{attribute 'no_explicit_call' := 'do not call this function block directly'} 
FUNCTION_BLOCK RenameFile EXTENDS ToolkitObject IMPLEMENTS IAction
VAR
	{attribute 'OPC.UA.DA' := '0'}
	_ClassName : STRING := __POUNAME();

	{attribute 'OPC.UA.DA' := '0'}
    _Rename : Tc2_System.FB_FileRename;
	
	{attribute 'OPC.UA.DA' := '0'}
	_NeedStart : BOOL;
	{attribute 'OPC.UA.DA' := '0'}
	_Done : BOOL;
END_VAR

{attribute 'monitoring' := 'call'}
{attribute 'OPC.UA.DA.Property' := '1'}
{attribute 'OPC.UA.DA' := '1'}
PROPERTY AmsNetId : Tc2_System.T_AmsNetID
GET
AmsNetId := _Rename.sNetId;
END_GET
SET
_Rename.sNetId := AmsNetId;
END_SET
END_PROPERTY

{attribute 'monitoring' := 'call'}
{attribute 'OPC.UA.DA.Property' := '1'}
{attribute 'OPC.UA.DA.Access' := '1'}
PROPERTY Busy : BOOL
GET
Busy := _NeedStart OR_ELSE _Rename.bBusy;
END_GET
END_PROPERTY

{attribute 'monitoring' := 'call'}
PROPERTY ClassName : STRING
GET
ClassName := _ClassName;
END_GET
END_PROPERTY

{attribute 'monitoring' := 'call'}
{attribute 'OPC.UA.DA.Property' := '1'}
{attribute 'OPC.UA.DA.Access' := '1'}
PROPERTY Done : BOOL
GET
Done := _Done;
END_GET
END_PROPERTY

{attribute 'monitoring' := 'call'}
{attribute 'OPC.UA.DA.Property' := '1'}
{attribute 'OPC.UA.DA.Access' := '1'}
PROPERTY Error : BOOL
GET
Error := _Rename.bError;
END_GET
END_PROPERTY

METHOD Execute
VAR
	message : ERROR_MESSAGE;
END_VAR
IF _NeedStart OR_ELSE _Rename.bBusy THEN
	_Rename(bExecute := TRUE);
	_NeedStart := FALSE;
	
	IF _Rename.bError THEN
		message := "An error occurred while renaming the file '";
		WStringHelper.Append6(message, TO_WSTRING(_Rename.sOldName), "' to '", TO_WSTRING(_Rename.sNewName), " in directory '", TO_WSTRING(_Rename.ePath), "'");	
		_LastException.Configure(message, __POUNAME(), ClassName, CurrentNamespace.Name, __POSITION(), _Rename.nErrId);
	ELSIF NOT _Rename.bBusy THEN
		_Done := TRUE;
	END_IF
END_IF
END_METHOD

{attribute 'monitoring' := 'call'}
{attribute 'OPC.UA.DA.Property' := '1'}
{attribute 'OPC.UA.DA.Access' := '1'}
PROPERTY LastException : REFERENCE TO Exception
GET
LastException REF= _LastException;
END_GET
END_PROPERTY

{attribute 'monitoring' := 'call'}
{attribute 'OPC.UA.DA.Property' := '1'}
{attribute 'OPC.UA.DA' := '1'}
PROPERTY PathType : Tc2_System.E_OpenPath
GET
PathType := _Rename.ePath;
END_GET
SET
_Rename.ePath := PathType;
END_SET
END_PROPERTY

METHOD Start
VAR_INPUT
	oldFilePath : Tc2_System.T_MaxString;
	newFilePath : Tc2_System.T_MaxString;
END_VAR
_NeedStart := TRUE;
_Done := FALSE;
_Rename.sOldName := oldFilePath;
_Rename.sNewName := newFilePath;

_LastException.Clear();
END_METHOD

{attribute 'monitoring' := 'call'}
{attribute 'OPC.UA.DA.Property' := '1'}
{attribute 'OPC.UA.DA' := '1'}
PROPERTY Timeout : TIME
GET
Timeout := _Rename.tTimeout;
END_GET
SET
_Rename.tTimeout := Timeout;
END_SET
END_PROPERTY

END_FUNCTION_BLOCK

(* stored: Version 1.1.0.1
   POU RenameFile: Id {c713f133-4ec6-4406-9624-5492aff6a30a}, SpecialFunc None
   Property AmsNetId: Id {aaebf810-5377-4278-8255-5fc10f6fd1a7}
   Get Get: Id {8f7f4a3b-e48f-48da-9fbf-90f8d00b12ac}
   Set Set: Id {fcef5c26-3ca6-4eb2-b89f-e16f4b09ad7b}
   Property Busy: Id {45c4f7c5-9da6-42a5-bc0e-5314f3d11305}
   Get Get: Id {82c0e643-96f5-4f46-8239-8bc96e2d619d}
   Property ClassName: Id {d4b42fdc-93bb-4ada-b91e-cd68aa93cd28}
   Get Get: Id {adf5bf3a-d6aa-405c-81a5-239df7314b9c}
   Property Done: Id {bfc87c89-79fc-45bc-b270-20c1045a8505}
   Get Get: Id {18b9f775-6886-4009-91c6-e8f3f71dd4c9}
   Property Error: Id {22240e1a-3239-41cf-9e1c-e932449a84d9}
   Get Get: Id {c0b5094f-d9dc-42f7-afff-aa6a9fd96631}
   Method Execute: Id {9c4f3b52-53f2-4442-a80d-985aba1c7574}
   Property LastException: Id {cd16af65-5f37-44a0-a3c1-ec6696fb9578}
   Get Get: Id {bc71fc19-048f-4675-94c9-153925cef64a}
   Property PathType: Id {f2b77e0e-ec2c-4d28-a222-f425245dd63c}
   Get Get: Id {ecf72d45-436f-4a95-8d9f-fe1246b3fc2c}
   Set Set: Id {fc7c92d6-8823-4161-955f-a38e61ebac19}
   Method Start: Id {54aa252f-bbc8-4b36-8268-eb691eedf8ae}
   Property Timeout: Id {6d64f9af-259f-45bf-b12b-566e9733abe0}
   Get Get: Id {4ed97089-387b-45e8-a712-823feee7213f}
   Set Set: Id {ee5bea57-ed6a-478e-9fe5-2f2a5ab6e0b0} *)
